// TIA Portal V20 export
TYPE "LER_typeCommunicationMonitoring"
// stored: Access Published
   STRUCT
      error : Bool;
      status : Word;
   END_STRUCT;
END_TYPE
